Omron Sysmac Studio project PeriodicTask_Uygulama (Sysmac Studio 1.65.0.64007, StandardProject)

# Controller new_Controller_0: NX1P2-1040DT1 version 1.69
Task PrimaryTask (priority 4, period or condition 2000): Program0
Task PeriodicTask0 (priority 17, period or condition 20000): Program1

VAR_GLOBAL RETAIN
    E_Set_Ramp : REAL;  (* published *)
    E_Max_Rpm : REAL;  (* published *)
    CycleTime : REAL;  (* published *)
    Stepp : REAL;  (* published *)
END_VAR
VAR_GLOBAL
    Ref_Rpm : REAL;  (* published *)
    Hizlan : BOOL;  (* published *)
    Yavasla : BOOL;  (* published *)
    Max_Rpm_Minus : REAL;  (* published *)
END_VAR

PROGRAM Program0

(* Section Section0: ladder, written here as Structured Text *)
END_PROGRAM

PROGRAM Program1
VAR_EXTERNAL
    Stepp : REAL;
    E_Max_Rpm : REAL;
    CycleTime : REAL;
    E_Set_Ramp : REAL;
    Max_Rpm_Minus : REAL;
    Hizlan : BOOL;
    Ref_Rpm : REAL;
    Yavasla : BOOL;
END_VAR

(* Section Section0: ladder, written here as Structured Text *)

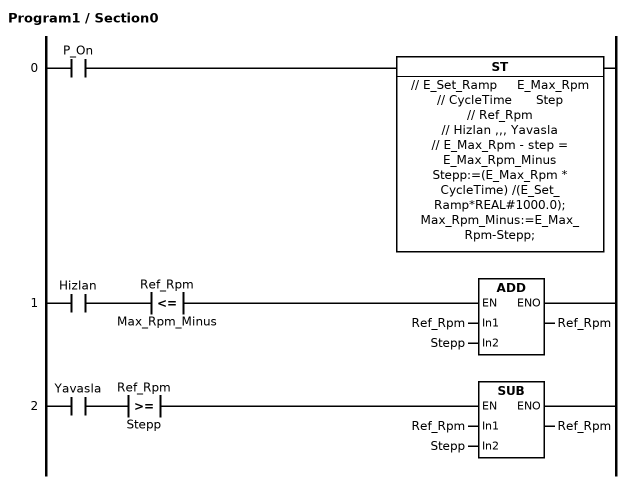
(* Rung 0 *)
IF P_On THEN
    // E_Set_Ramp			E_Max_Rpm
    // CycleTime			Step
    // Ref_Rpm
    // Hizlan ,,, Yavasla
    // E_Max_Rpm - step = E_Max_Rpm_Minus
    Stepp:=(E_Max_Rpm * CycleTime) /(E_Set_Ramp*REAL#1000.0);
    Max_Rpm_Minus:=E_Max_Rpm-Stepp;
END_IF;
(* Rung 1 *)
IF Hizlan AND (Ref_Rpm <= Max_Rpm_Minus) THEN Ref_Rpm := Ref_Rpm + Stepp; END_IF;
(* Rung 2 *)
IF Yavasla AND (Ref_Rpm >= Stepp) THEN Ref_Rpm := Ref_Rpm - Stepp; END_IF;
END_PROGRAM